FUNCTION_BLOCK IAS_SKILL_DEMUX_GEN (* Composite Function Block Type *)
  (* Standard: 61499-2 *)
  (* Version 0.0, 2008-07-10, 4DIAC-IDE, 4DIAC-Consortium *)
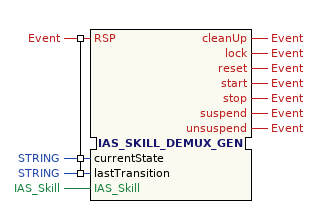
  EVENT_INPUT
    RSP WITH currentState, lastTransition;
  END_EVENT
  EVENT_OUTPUT
    cleanUp;
    lock;
    reset;
    start;
    stop;
    suspend;
    unsuspend;
  END_EVENT
  VAR_INPUT
    currentState : STRING;
    lastTransition : STRING;
  END_VAR
  SOCKETS
    IAS_Skill : IAS_Skill;
  END_SOCKETS
  EVENT_CONNECTIONS
    RSP TO IAS_Skill.RSP;
    IAS_Skill.cleanUp TO cleanUp;
    IAS_Skill.lock TO lock;
    IAS_Skill.reset TO reset;
    IAS_Skill.start TO start;
    IAS_Skill.stop TO stop;
    IAS_Skill.suspend TO suspend;
    IAS_Skill.unsuspend TO unsuspend;
  END_CONNECTIONS
  DATA_CONNECTIONS
    currentState TO IAS_Skill.currentState;
    lastTransition TO IAS_Skill.lastTransition;
  END_CONNECTIONS
END_FUNCTION_BLOCK
